INTERFACE I_LinearEncodedDrive EXTENDS I_LinearContinuousDrive, I_EncodedDrive

END_INTERFACE

(* stored: Version 1.1.0.1, ProductVersion 3.1.4024.11
   Itf I_LinearEncodedDrive: Id {7174a65f-c6cc-446f-9555-70fb88afef07} *)
